// LS Electric XG5000 project: #1_1
// PLC NewPLC

PROGRAM NewProgram (task: 스캔 프로그램)

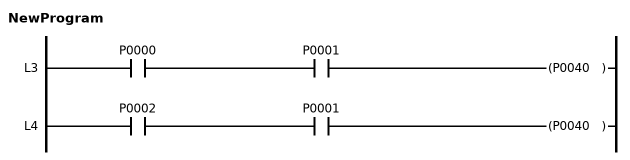
; L3
LOAD      P0000
AND       P0001
OUT       P0040
; L4
LOAD      P0002
AND       P0001
OUT       P0040